INTERFACE I_PersistentEventStorage

METHOD StoreEvent 
VAR_INPUT
	stEvent : St_Event ;
	
END_VAR
END_METHOD

END_INTERFACE

(* stored: Version 1.1.0.1, ProductVersion 3.1.4024.12
   Itf I_PersistentEventStorage: Id {3b6e8ae5-8938-40f0-9ecd-7c4aee4851f8}
   Method StoreEvent: Id {6c6a90bf-41ac-4da0-9780-597ca11dcc9b} *)
